TYPE "SpeedMachine_Alr"
VERSION : 0.1
// Block: SpeedMachine_Alr
   STRUCT
      BrakeTimeOut : Bool;
      S120_ComErr : Bool;
      Ax : Struct
         Drive : Bool;
      END_STRUCT;
      Fan_M : MotorAlr;
   END_STRUCT;

END_TYPE
